// TIA Portal project "Ejemplo_4" (V16)

(* hardware
DEVICE "S7300/ET200M station_1"  S7-300 station
   slot 0: "Perfil soporte_0"  Rail  6ES7 390-1***0-0AA0
   slot 2: "PLC_1"  CPU 313C  6ES7 313-5BG04-0AB0  V3.3
      slot 0: "Interfaz MPI_1"  MPI
      slot 2: "DI 24/DO 16_1"  DI24/DO16
      slot 3: "AI 5/AO 2_1"  AI5/AO2
      slot 4: "Contaje_1"  Counter
   slot 4: "CP 343-1 Lean_1"  CP 343-1 LEAN  6GK7 343-1CX10-0XE0  V3.0
DEVICE "HMI_1"  KTP1000 Basic color DP
   slot 0: "HMI_1"  KTP1000 Basic color DP  6AV6 647-0AE11-3AX0  12.0.0.0
   slot 1: "HMI_RT_1"  KTP1000 Basic color DP  6AV6 647-0AE11-3AX0  12.0.0.0
   slot 7: "HMI_1.MPI/DP_CP_1"  MPI/DP Interface  12.0.0.0
*)

// ===== PLC "PLC_1"  CPU 313C =====

VAR_GLOBAL   // PLC tag table "Tabla de variables estándar"
   "Tag_2" AT %I124.0 : Bool;
   "Tag_3" AT %Q124.0 : Bool;
   "ADC" AT %IW752 : Int;
   "MADC" AT %MW0 : Int;
END_VAR

DATA_BLOCK "Variables"   // DB1
{ S7_Optimized_Access := 'FALSE' }
VERSION : 0.1
   VAR
      Boton : Bool;
      Potenciometro : Int;
      Led : Bool;
      Sensor : Real;
   END_VAR
BEGIN
END_DATA_BLOCK

ORGANIZATION_BLOCK "Main"   // OB1, LAD
TITLE = "Main Program Sweep (Cycle)"
{ S7_Optimized_Access := 'FALSE' }
VERSION : 0.1
   VAR_TEMP
      OB1_EV_CLASS : Byte;   // Bits 0-3 = 1 (Coming event), Bits 4-7 = 1 (Event class 1)
      OB1_SCAN_1 : Byte;   // 1 (Cold restart scan 1 of OB 1), 3 (Scan 2-n of OB 1)
      OB1_PRIORITY : Byte;   // Priority of OB Execution
      OB1_OB_NUMBR : Byte;   // 1 (Organization block 1, OB1)
      OB1_RESERVED_1 : Byte;   // Reserved for system
      OB1_RESERVED_2 : Byte;   // Reserved for system
      OB1_PREV_CYCLE : Int;   // Cycle time of previous OB1 scan (milliseconds)
      OB1_MIN_CYCLE : Int;   // Minimum cycle time of OB1 (milliseconds)
      OB1_MAX_CYCLE : Int;   // Maximum cycle time of OB1 (milliseconds)
      OB1_DATE_TIME : Date_And_Time;   // Date and time OB1 started
      Flag : Bool;
      Error : Word;
   END_VAR
BEGIN

REGION Network 1
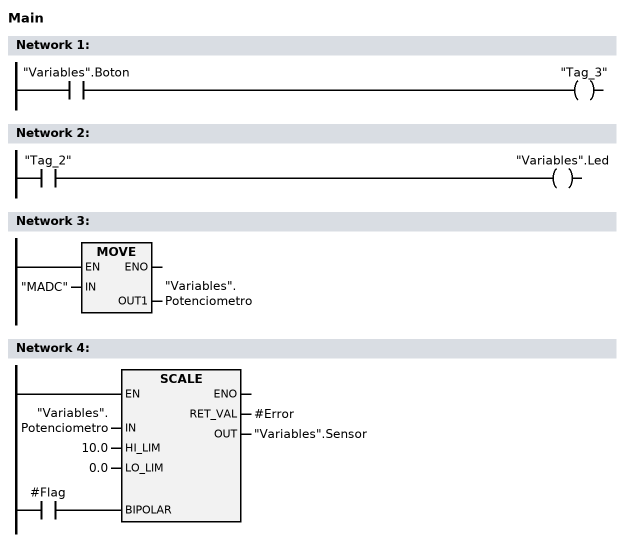
   RUNG wire#powerrail
      Contact( "Variables".Boton )
      Coil( "Tag_3" )
   END_RUNG
   // the same network as SCL:
   "Tag_3" := "Variables".Boton;
END_REGION

REGION Network 2
   RUNG wire#powerrail
      Contact( "Tag_2" )
      Coil( "Variables".Led )
   END_RUNG
   // the same network as SCL:
   "Variables".Led := "Tag_2";
END_REGION

REGION Network 3
   RUNG wire#powerrail
      { S7_GenerateENO := "TRUE" } Move(in := "MADC", out1 => "Variables".Potenciometro)
   END_RUNG
   // the same network as SCL:
   "Variables".Potenciometro := "MADC";
END_REGION

REGION Network 4
   #Error := SCALE(IN := "Variables".Potenciometro,
                   HI_LIM := 10.0,
                   LO_LIM := 0.0,
                   BIPOLAR := #Flag,
                   OUT => "Variables".Sensor);
END_REGION
END_ORGANIZATION_BLOCK

(* ===== HMI "HMI_RT_1" =====
system functions are stored by id; their names below are inferred from use
connection "HMI_Conexión_1": IF1 B, SIMATIC S7 300/400 MPI

HMI tags "Tabla de variables estándar"
   "Número_imagen_variable" : UInt, internal
   "Variables_Boton" : Bool = PLC Variables.Boton AT %DB1.DBX0.0, 1 s
   "Tag_3" : Bool = PLC Tag_3 AT %Q124.0, 1 s

text list "Nombre_imagen_lista_texto": 1 'Imagen raíz'

Template "Plantilla_1" 640x480
   Button "Salir" at 560,422 size 79x57; TextOff 'Salir'; PictureOff "ExitRuntime_KTP1000_Basic_color_DP"; PictureOn "ExitRuntime_KTP1000_Basic_color_DP"
      on Release: StopRuntime(0)
   Button "Template_Button" at 480,422 size 79x57; TextOff 'Text'
   Button "Template_Button_1" at 400,422 size 79x57; TextOff 'Text'
   Button "Template_Button_2" at 320,422 size 79x57; TextOff 'Text'
   Button "Template_Button_3" at 240,422 size 79x57; TextOff 'Text'
   Button "Template_Button_4" at 160,422 size 79x57; TextOff 'Text'
   Button "Template_Button_5" at 80,422 size 79x57; TextOff 'Text'
   Button "Imagen inicial" at 0,422 size 79x57; TextOff 'Imagen inicial'; PictureOff "NavigateHome_KTP1000_Basic_color_DP"; PictureOn "NavigateHome_KTP1000_Basic_color_DP"
      on Release: ActivateScreen("Imagen raíz", 0)
   SymbolicIOField "Imagen_campo_ES_simbólico" at 105,11 size 428x34; TextOff '0'; TextOn '1'; TextList "Nombre_imagen_lista_texto"
      ProcessValue <- "Número_imagen_variable"
      on Change: ActivateScreenByNumber("Número_imagen_variable", 0)
   DateTimeField "HmiScreenItemData" at 535,29 size 105x29
   DateTimeField "HmiScreenItemData_1" at 535,0 size 105x29
   GraphicView "Logotipo" at 0,0 size 103x58; Picture "Logotipo de HMI_1"

screen "Imagen raíz" 640x480, template "Plantilla_1"
   on GenerateScreen: SetTag("Número_imagen_variable", 1)
   Circle "Círculo_1" at 388,164 size 48x48
      Appearance <- "Tag_3"
   Button "Botón_1" at 171,175 size 96x32; TextOff 'Invertir'
      on Press: InvertBit("Variables_Boton")
   Bar "Barra_1" at 491,107 size 100x200; MinimumValue 0; MaximumValue 100
*)